(* PLC project ST_CALL_BASIC.project, Inovance company InoProShop(V1.8.1.3) InoProShop(V1.8.1.3) *)
(* stored: creationDateTime 2025-03-20T13:33:35.5388734, modificationDateTime 2025-03-19T17:06:50.1361953 *)

PROGRAM PLC_PRG
  VAR
    cur : INT;
    out1 : INT;
    FB00 : FB0;
    var1 : INT;
    bool1 : BOOL;
  END_VAR

                  FB00();

IF con1 THEN
FB00();
END_IF;
var1:=1;
var1:=var1*3;
func (in1:=bool1);

                
END_PROGRAM

FUNCTION_BLOCK FB0
  VAR
    out1 : INT;
    TON0 : TON;
  END_VAR

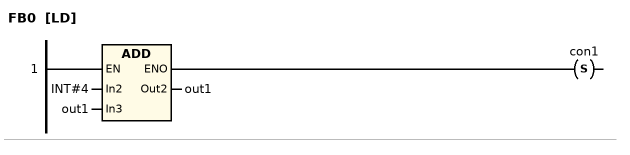
(* LD diagram, written out as Structured Text *)
(* 网络注释 *)

out1 := INT#4 + out1;
IF TRUE THEN con1 := TRUE; END_IF;
END_FUNCTION_BLOCK

PROGRAM func
  VAR
    TON0 : TON;
  END_VAR
  VAR_INPUT
    in1 : BOOL;
  END_VAR

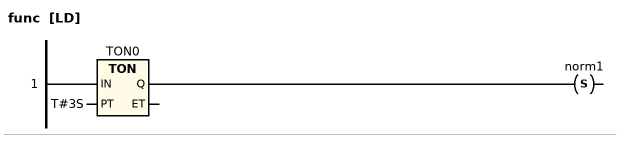
(* LD diagram, written out as Structured Text *)
(* 网络注释 *)

TON0(IN := TRUE, PT := T#3S);
IF TON0.Q THEN norm1 := TRUE; END_IF;
END_PROGRAM

CONFIGURATION Application
  RESOURCE Application ON PLC
    VAR_GLOBAL RETAIN PERSISTENT  (* GVL *)
      con1 AT %MB131072 : BOOL := TRUE;
      con2 : BOOL;
      norm1 : BOOL;
    END_VAR
  END_RESOURCE
END_CONFIGURATION
